Universal Robots PolyScope program: GlobalToLocal.urp

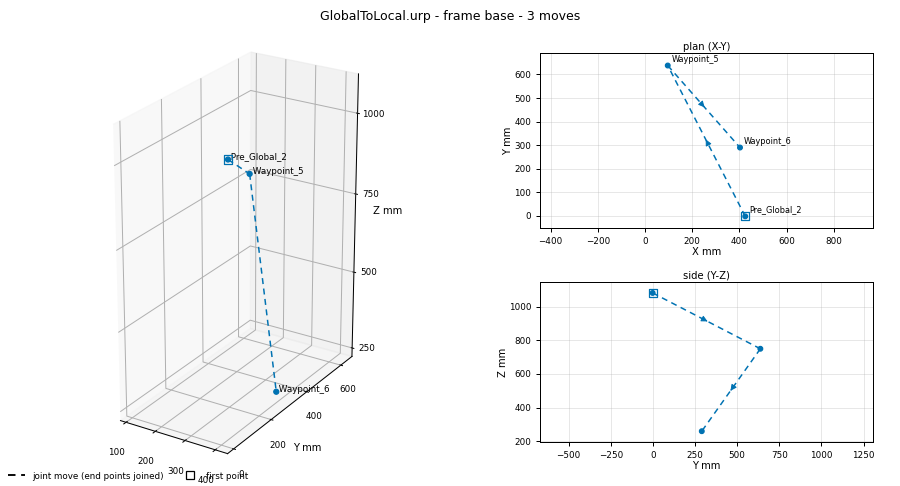
[picture p0: tool path of GlobalToLocal.urp in frame base, 3 of 4 moves have a stored position in this frame; points joined in program order, loops and branches not executed]
Program GlobalToLocal (installation=Youssef directory=/programs/Youssef createdIn=5.9.5.1031259 lastSavedIn=5.9.5.1031259 robotSerialNumber=20215500597)
Calibrated DH parameters: a=[0.000193, -0.066673, -0.391568, -0.000012, 0.00005, 0]; d=[0.162643, -472.05677, 465.132521, 7.058239, 0.099746, 0.099582]; alpha=[1.571116, 0.00089, 0.003862, 1.569269, -1.569248, 0]; deltaTheta=[0, -1.413394, 7.628392, 0.068187, 0, -0.000001]
Robot Program (runOnlyOnce=true)
  MoveJ speed 60 deg/s, acceleration 80 deg/s^2 (useActiveTCP=true) feature=Base
    SafeHome (positionOptionType=SPEED_AND_ACCELERATION speed=1.047198 acceleration=1.396263 nextMotionTime=2)
    Waypoint Pre_Global_2: TCP in base x=424.817 y=-1.551 z=1080.554 mm, rx=-1.2067 ry=1.2116 rz=-1.2125 rad; joints [89.999, -90, 0, -89.996, -0.001, -0.002] deg; TCP offset x=0 y=0 z=191.5 mm, rx=0 ry=0 rz=0 rad
    Waypoint Waypoint_5: TCP in base x=96.27 y=637.775 z=749.236 mm, rx=-1.4855 ry=-0.0307 rz=0.0319 rad; joints [94.292, -84.133, -90.199, -0.883, 88.027, -0.054] deg
    Waypoint Waypoint_6: TCP in base x=402.516 y=290.095 z=259.958 mm, rx=1.3002 ry=1.1489 rz=1.2399 rad; joints [94.435, -83.523, -131.099, -136.444, 6.698, -3.896] deg
    Waypoint Waypoint (Variable): variable(featureName=Local)
